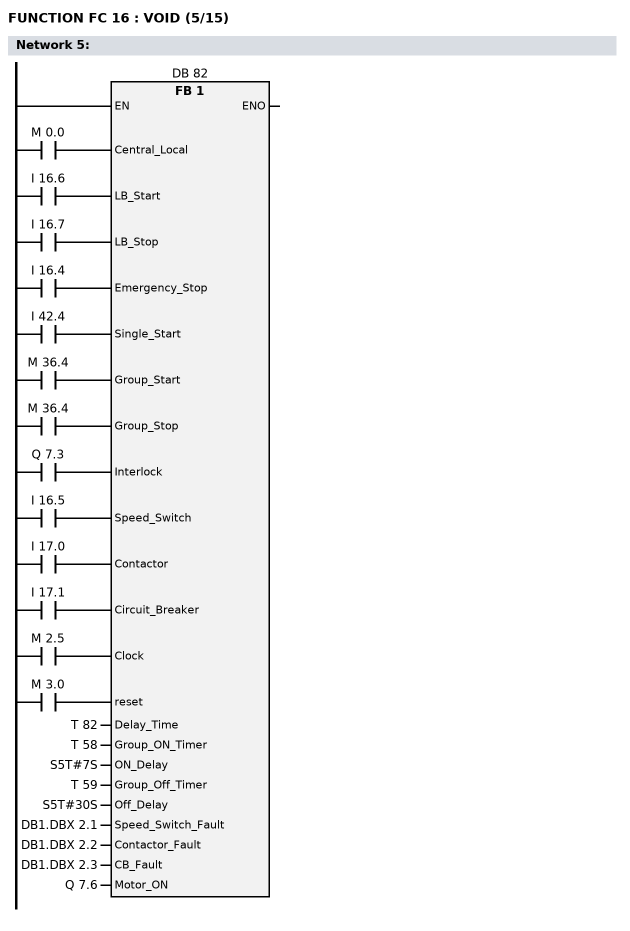

      A     M      0.0;
      =     L      0.0;
      BLD   103;
      A     I     16.6;
      =     L      0.1;
      BLD   103;
      A     I     16.7;
      =     L      0.2;
      BLD   103;
      A     I     16.4;
      =     L      0.3;
      BLD   103;
      A     I     42.4;
      =     L      0.4;
      BLD   103;
      A     M     36.4;
      =     L      0.5;
      BLD   103;
      A     M     36.4;
      =     L      0.6;
      BLD   103;
      A     Q      7.3;
      =     L      0.7;
      BLD   103;
      A     I     16.5;
      =     L      1.0;
      BLD   103;
      A     I     17.0;
      =     L      1.1;
      BLD   103;
      A     I     17.1;
      =     L      1.2;
      BLD   103;
      A     M      2.5;
      =     L      1.3;
      BLD   103;
      A     M      3.0;
      =     L      1.4;
      BLD   103;
      CALL FB     1 , DB    82 (
           Central_Local            := L      0.0,
           LB_Start                 := L      0.1,
           LB_Stop                  := L      0.2,
           Emergency_Stop           := L      0.3,
           Single_Start             := L      0.4,
           Group_Start              := L      0.5,
           Group_Stop               := L      0.6,
           Interlock                := L      0.7,
           Speed_Switch             := L      1.0,
           Contactor                := L      1.1,
           Circuit_Breaker          := L      1.2,
           Clock                    := L      1.3,
           reset                    := L      1.4,
           Delay_Time               := T     82,
           Group_ON_Timer           := T     58,
           ON_Delay                 := S5T#7S,
           Group_Off_Timer          := T     59,
           Off_Delay                := S5T#30S,
           Speed_Switch_Fault       := DB1.DBX    2.1,
           Contactor_Fault          := DB1.DBX    2.2,
           CB_Fault                 := DB1.DBX    2.3,
           Motor_ON                 := Q      7.6);
      NOP   0;
NETWORK
TITLE =
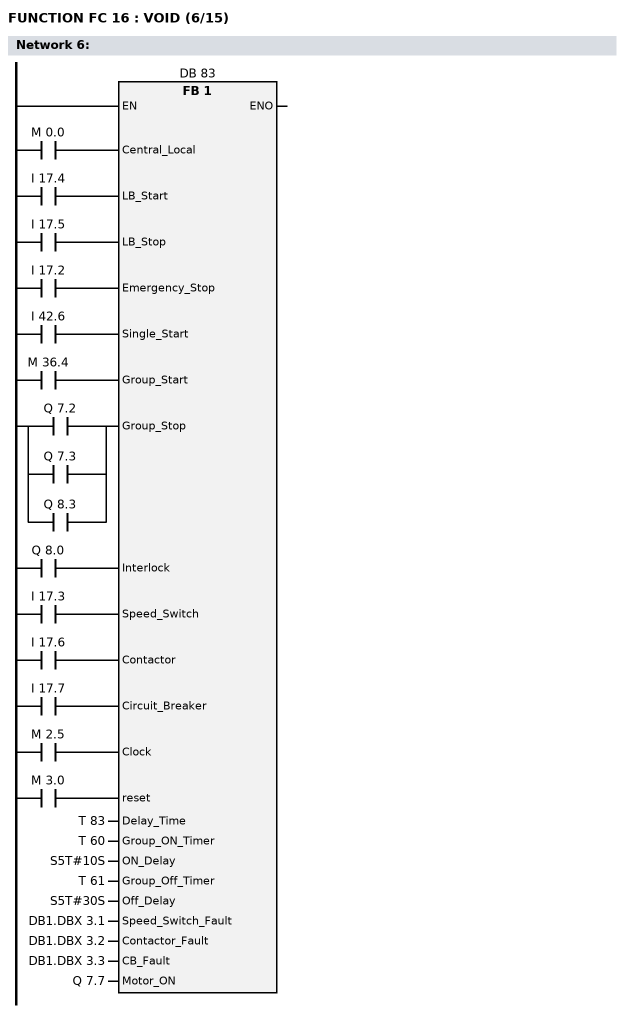

      A     M      0.0;
      =     L      0.0;
      BLD   103;
      A     I     17.4;
      =     L      0.1;
      BLD   103;
      A     I     17.5;
      =     L      0.2;
      BLD   103;
      A     I     17.2;
      =     L      0.3;
      BLD   103;
      A     I     42.6;
      =     L      0.4;
      BLD   103;
      A     M     36.4;
      =     L      0.5;
      BLD   103;
      A(    ;
      O     Q      7.2;
      O     Q      7.3;
      O     Q      8.3;
      )     ;
      =     L      0.6;
      BLD   103;
      A     Q      8.0;
      =     L      0.7;
      BLD   103;
      A     I     17.3;
      =     L      1.0;
      BLD   103;
      A     I     17.6;
      =     L      1.1;
      BLD   103;
      A     I     17.7;
      =     L      1.2;
      BLD   103;
      A     M      2.5;
      =     L      1.3;
      BLD   103;
      A     M      3.0;
      =     L      1.4;
      BLD   103;
      CALL FB     1 , DB    83 (
           Central_Local            := L      0.0,
           LB_Start                 := L      0.1,
           LB_Stop                  := L      0.2,
           Emergency_Stop           := L      0.3,
           Single_Start             := L      0.4,
           Group_Start              := L      0.5,
           Group_Stop               := L      0.6,
           Interlock                := L      0.7,
           Speed_Switch             := L      1.0,
           Contactor                := L      1.1,
           Circuit_Breaker          := L      1.2,
           Clock                    := L      1.3,
           reset                    := L      1.4,
           Delay_Time               := T     83,
           Group_ON_Timer           := T     60,
           ON_Delay                 := S5T#10S,
           Group_Off_Timer          := T     61,
           Off_Delay                := S5T#30S,
           Speed_Switch_Fault       := DB1.DBX    3.1,
           Contactor_Fault          := DB1.DBX    3.2,
           CB_Fault                 := DB1.DBX    3.3,
           Motor_ON                 := Q      7.7);
      NOP   0;
NETWORK
TITLE =
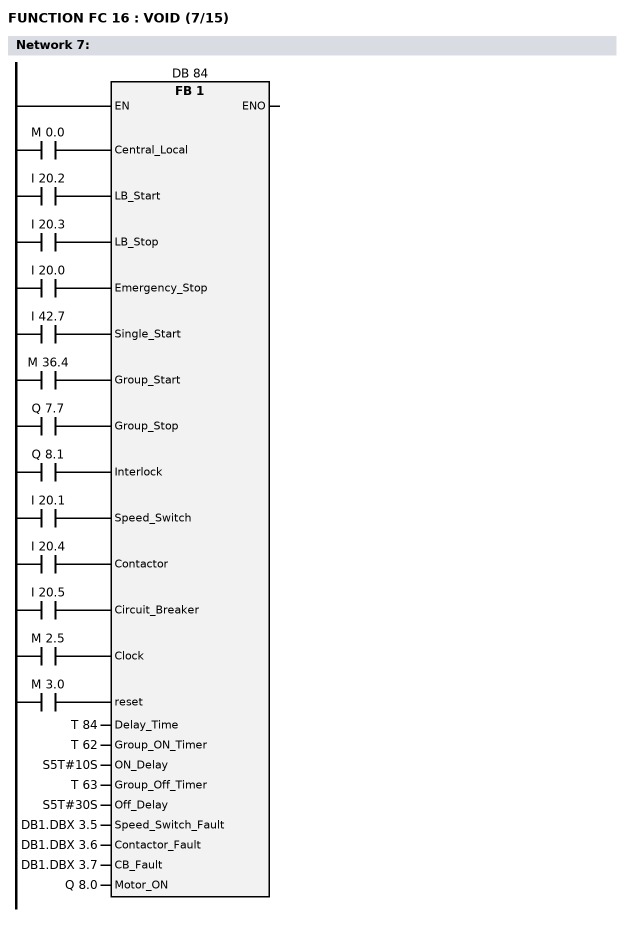

      A     M      0.0;
      =     L      0.0;
      BLD   103;
      A     I     20.2;
      =     L      0.1;
      BLD   103;
      A     I     20.3;
      =     L      0.2;
      BLD   103;
      A     I     20.0;
      =     L      0.3;
      BLD   103;
      A     I     42.7;
      =     L      0.4;
      BLD   103;
      A     M     36.4;
      =     L      0.5;
      BLD   103;
      A     Q      7.7;
      =     L      0.6;
      BLD   103;
      A     Q      8.1;
      =     L      0.7;
      BLD   103;
      A     I     20.1;
      =     L      1.0;
      BLD   103;
      A     I     20.4;
      =     L      1.1;
      BLD   103;
      A     I     20.5;
      =     L      1.2;
      BLD   103;
      A     M      2.5;
      =     L      1.3;
      BLD   103;
      A     M      3.0;
      =     L      1.4;
      BLD   103;
      CALL FB     1 , DB    84 (
           Central_Local            := L      0.0,
           LB_Start                 := L      0.1,
           LB_Stop                  := L      0.2,
           Emergency_Stop           := L      0.3,
           Single_Start             := L      0.4,
           Group_Start              := L      0.5,
           Group_Stop               := L      0.6,
           Interlock                := L      0.7,
           Speed_Switch             := L      1.0,
           Contactor                := L      1.1,
           Circuit_Breaker          := L      1.2,
           Clock                    := L      1.3,
           reset                    := L      1.4,
           Delay_Time               := T     84,
           Group_ON_Timer           := T     62,
           ON_Delay                 := S5T#10S,
           Group_Off_Timer          := T     63,
           Off_Delay                := S5T#30S,
           Speed_Switch_Fault       := DB1.DBX    3.5,
           Contactor_Fault          := DB1.DBX    3.6,
           CB_Fault                 := DB1.DBX    3.7,
           Motor_ON                 := Q      8.0);
      NOP   0;
NETWORK
TITLE =
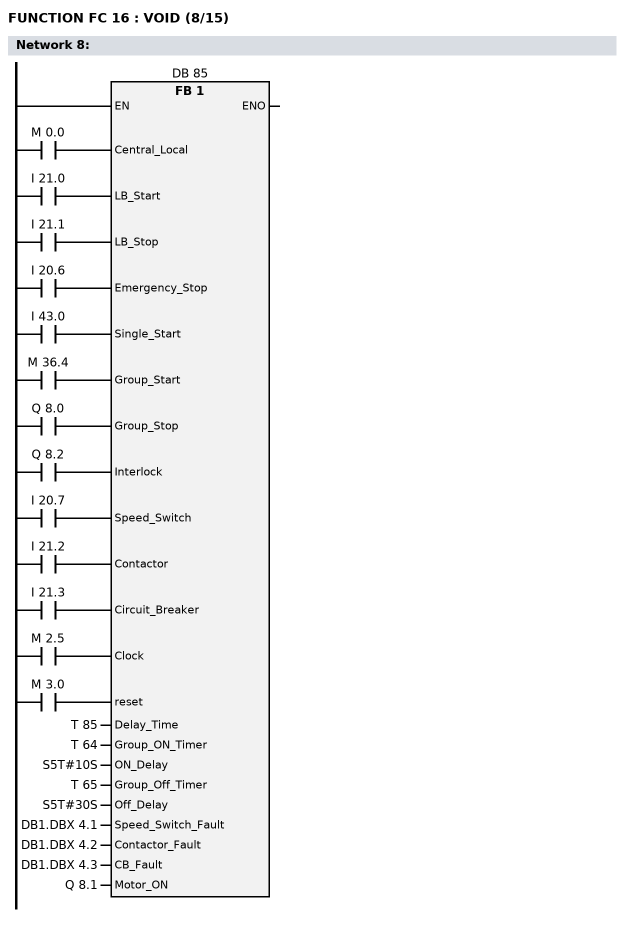

      A     M      0.0;
      =     L      0.0;
      BLD   103;
      A     I     21.0;
      =     L      0.1;
      BLD   103;
      A     I     21.1;
      =     L      0.2;
      BLD   103;
      A     I     20.6;
      =     L      0.3;
      BLD   103;
      A     I     43.0;
      =     L      0.4;
      BLD   103;
      A     M     36.4;
      =     L      0.5;
      BLD   103;
      A     Q      8.0;
      =     L      0.6;
      BLD   103;
      A     Q      8.2;
      =     L      0.7;
      BLD   103;
      A     I     20.7;
      =     L      1.0;
      BLD   103;
      A     I     21.2;
      =     L      1.1;
      BLD   103;
      A     I     21.3;
      =     L      1.2;
      BLD   103;
      A     M      2.5;
      =     L      1.3;
      BLD   103;
      A     M      3.0;
      =     L      1.4;
      BLD   103;
      CALL FB     1 , DB    85 (
           Central_Local            := L      0.0,
           LB_Start                 := L      0.1,
           LB_Stop                  := L      0.2,
           Emergency_Stop           := L      0.3,
           Single_Start             := L      0.4,
           Group_Start              := L      0.5,
           Group_Stop               := L      0.6,
           Interlock                := L      0.7,
           Speed_Switch             := L      1.0,
           Contactor                := L      1.1,
           Circuit_Breaker          := L      1.2,
           Clock                    := L      1.3,
           reset                    := L      1.4,
           Delay_Time               := T     85,
           Group_ON_Timer           := T     64,
           ON_Delay                 := S5T#10S,
           Group_Off_Timer          := T     65,
           Off_Delay                := S5T#30S,
           Speed_Switch_Fault       := DB1.DBX    4.1,
           Contactor_Fault          := DB1.DBX    4.2,
           CB_Fault                 := DB1.DBX    4.3,
           Motor_ON                 := Q      8.1);
      NOP   0;
NETWORK
TITLE =
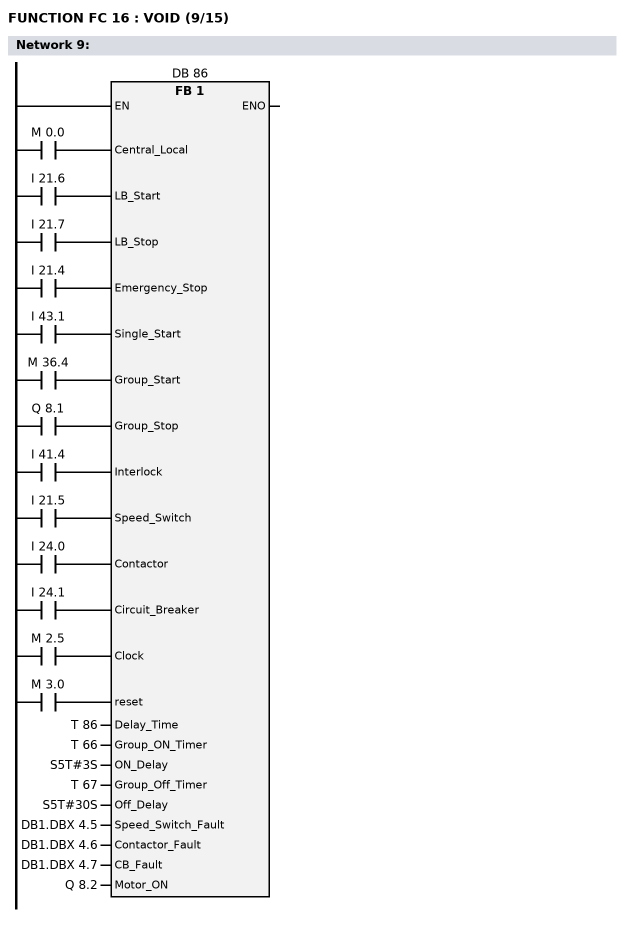

      A     M      0.0;
      =     L      0.0;
      BLD   103;
      A     I     21.6;
      =     L      0.1;
      BLD   103;
      A     I     21.7;
      =     L      0.2;
      BLD   103;
      A     I     21.4;
      =     L      0.3;
      BLD   103;
      A     I     43.1;
      =     L      0.4;
      BLD   103;
      A     M     36.4;
      =     L      0.5;
      BLD   103;
      A     Q      8.1;
      =     L      0.6;
      BLD   103;
      A     I     41.4;
      =     L      0.7;
      BLD   103;
      A     I     21.5;
      =     L      1.0;
      BLD   103;
      A     I     24.0;
      =     L      1.1;
      BLD   103;
      A     I     24.1;
      =     L      1.2;
      BLD   103;
      A     M      2.5;
      =     L      1.3;
      BLD   103;
      A     M      3.0;
      =     L      1.4;
      BLD   103;
      CALL FB     1 , DB    86 (
           Central_Local            := L      0.0,
           LB_Start                 := L      0.1,
           LB_Stop                  := L      0.2,
           Emergency_Stop           := L      0.3,
           Single_Start             := L      0.4,
           Group_Start              := L      0.5,
           Group_Stop               := L      0.6,
           Interlock                := L      0.7,
           Speed_Switch             := L      1.0,
           Contactor                := L      1.1,
           Circuit_Breaker          := L      1.2,
           Clock                    := L      1.3,
           reset                    := L      1.4,
           Delay_Time               := T     86,
           Group_ON_Timer           := T     66,
           ON_Delay                 := S5T#3S,
           Group_Off_Timer          := T     67,
           Off_Delay                := S5T#30S,
           Speed_Switch_Fault       := DB1.DBX    4.5,
           Contactor_Fault          := DB1.DBX    4.6,
           CB_Fault                 := DB1.DBX    4.7,
           Motor_ON                 := Q      8.2);
      NOP   0;
NETWORK
TITLE =
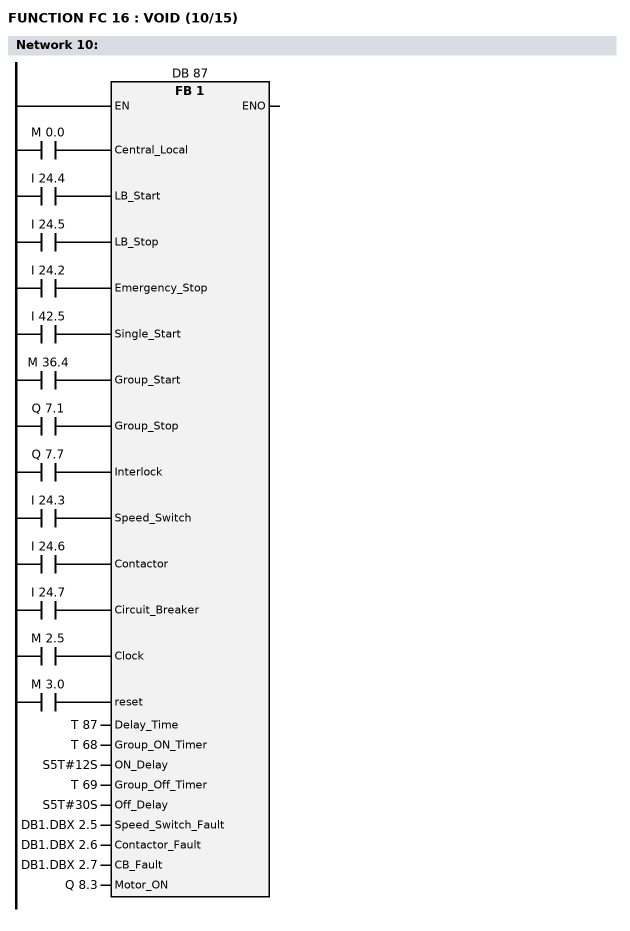

      A     M      0.0;
      =     L      0.0;
      BLD   103;
      A     I     24.4;
      =     L      0.1;
      BLD   103;
      A     I     24.5;
      =     L      0.2;
      BLD   103;
      A     I     24.2;
      =     L      0.3;
      BLD   103;
      A     I     42.5;
      =     L      0.4;
      BLD   103;
      A     M     36.4;
      =     L      0.5;
      BLD   103;
      A     Q      7.1;
      =     L      0.6;
      BLD   103;
      A     Q      7.7;
      =     L      0.7;
      BLD   103;
      A     I     24.3;
      =     L      1.0;
      BLD   103;
      A     I     24.6;
      =     L      1.1;
      BLD   103;
      A     I     24.7;
      =     L      1.2;
      BLD   103;
      A     M      2.5;
      =     L      1.3;
      BLD   103;
      A     M      3.0;
      =     L      1.4;
      BLD   103;
      CALL FB     1 , DB    87 (
           Central_Local            := L      0.0,
           LB_Start                 := L      0.1,
           LB_Stop                  := L      0.2,
           Emergency_Stop           := L      0.3,
           Single_Start             := L      0.4,
           Group_Start              := L      0.5,
           Group_Stop               := L      0.6,
           Interlock                := L      0.7,
           Speed_Switch             := L      1.0,
           Contactor                := L      1.1,
           Circuit_Breaker          := L      1.2,
           Clock                    := L      1.3,
           reset                    := L      1.4,
           Delay_Time               := T     87,
           Group_ON_Timer           := T     68,
           ON_Delay                 := S5T#12S,
           Group_Off_Timer          := T     69,
           Off_Delay                := S5T#30S,
           Speed_Switch_Fault       := DB1.DBX    2.5,
           Contactor_Fault          := DB1.DBX    2.6,
           CB_Fault                 := DB1.DBX    2.7,
           Motor_ON                 := Q      8.3);
      NOP   0;
NETWORK
TITLE =
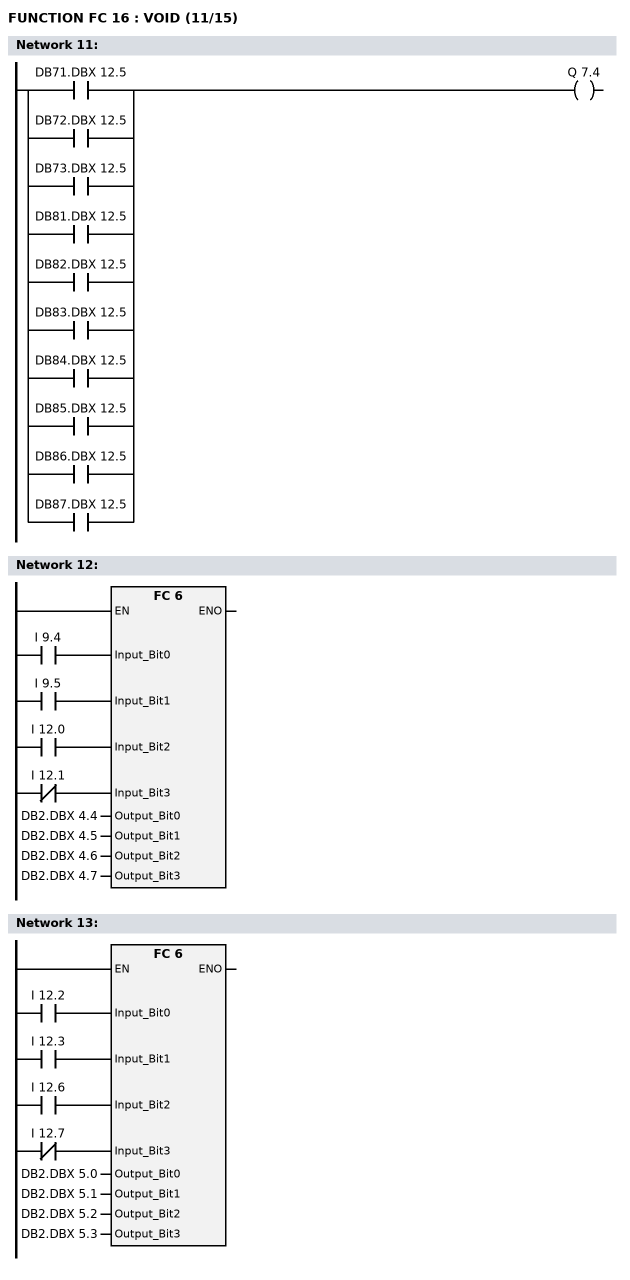

      O     DB71.DBX   12.5;
      O     DB72.DBX   12.5;
      O     DB73.DBX   12.5;
      O     DB81.DBX   12.5;
      O     DB82.DBX   12.5;
      O     DB83.DBX   12.5;
      O     DB84.DBX   12.5;
      O     DB85.DBX   12.5;
      O     DB86.DBX   12.5;
      O     DB87.DBX   12.5;
      =     Q      7.4;
NETWORK
TITLE =

      A     I      9.4;
      =     L      0.0;
      BLD   103;
      A     I      9.5;
      =     L      0.1;
      BLD   103;
      A     I     12.0;
      =     L      0.2;
      BLD   103;
      AN    I     12.1;
      =     L      0.3;
      BLD   103;
      CALL FC     6 (
           Input_Bit0               := L      0.0,
           Input_Bit1               := L      0.1,
           Input_Bit2               := L      0.2,
           Input_Bit3               := L      0.3,
           Output_Bit0              := DB2.DBX    4.4,
           Output_Bit1              := DB2.DBX    4.5,
           Output_Bit2              := DB2.DBX    4.6,
           Output_Bit3              := DB2.DBX    4.7);
      NOP   0;
NETWORK
TITLE =

      A     I     12.2;
      =     L      0.0;
      BLD   103;
      A     I     12.3;
      =     L      0.1;
      BLD   103;
      A     I     12.6;
      =     L      0.2;
      BLD   103;
      AN    I     12.7;
      =     L      0.3;
      BLD   103;
      CALL FC     6 (
           Input_Bit0               := L      0.0,
           Input_Bit1               := L      0.1,
           Input_Bit2               := L      0.2,
           Input_Bit3               := L      0.3,
           Output_Bit0              := DB2.DBX    5.0,
           Output_Bit1              := DB2.DBX    5.1,
           Output_Bit2              := DB2.DBX    5.2,
           Output_Bit3              := DB2.DBX    5.3);
      NOP   0;
NETWORK
TITLE =
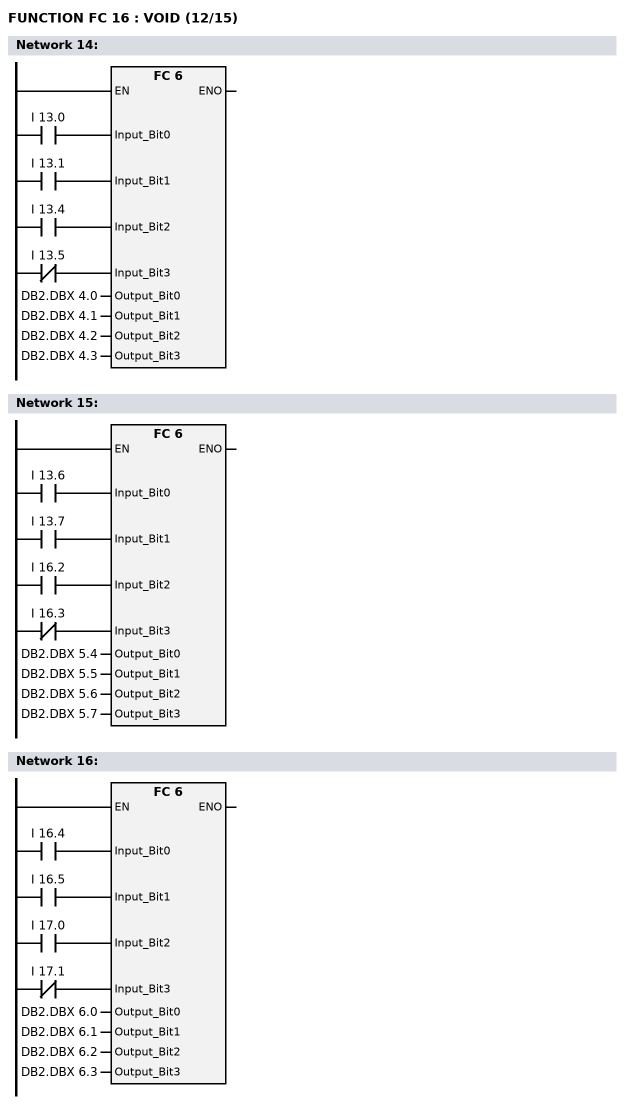

      A     I     13.0;
      =     L      0.0;
      BLD   103;
      A     I     13.1;
      =     L      0.1;
      BLD   103;
      A     I     13.4;
      =     L      0.2;
      BLD   103;
      AN    I     13.5;
      =     L      0.3;
      BLD   103;
      CALL FC     6 (
           Input_Bit0               := L      0.0,
           Input_Bit1               := L      0.1,
           Input_Bit2               := L      0.2,
           Input_Bit3               := L      0.3,
           Output_Bit0              := DB2.DBX    4.0,
           Output_Bit1              := DB2.DBX    4.1,
           Output_Bit2              := DB2.DBX    4.2,
           Output_Bit3              := DB2.DBX    4.3);
      NOP   0;
NETWORK
TITLE =

      A     I     13.6;
      =     L      0.0;
      BLD   103;
      A     I     13.7;
      =     L      0.1;
      BLD   103;
      A     I     16.2;
      =     L      0.2;
      BLD   103;
      AN    I     16.3;
      =     L      0.3;
      BLD   103;
      CALL FC     6 (
           Input_Bit0               := L      0.0,
           Input_Bit1               := L      0.1,
           Input_Bit2               := L      0.2,
           Input_Bit3               := L      0.3,
           Output_Bit0              := DB2.DBX    5.4,
           Output_Bit1              := DB2.DBX    5.5,
           Output_Bit2              := DB2.DBX    5.6,
           Output_Bit3              := DB2.DBX    5.7);
      NOP   0;
NETWORK
TITLE =

      A     I     16.4;
      =     L      0.0;
      BLD   103;
      A     I     16.5;
      =     L      0.1;
      BLD   103;
      A     I     17.0;
      =     L      0.2;
      BLD   103;
      AN    I     17.1;
      =     L      0.3;
      BLD   103;
      CALL FC     6 (
           Input_Bit0               := L      0.0,
           Input_Bit1               := L      0.1,
           Input_Bit2               := L      0.2,
           Input_Bit3               := L      0.3,
           Output_Bit0              := DB2.DBX    6.0,
           Output_Bit1              := DB2.DBX    6.1,
           Output_Bit2              := DB2.DBX    6.2,
           Output_Bit3              := DB2.DBX    6.3);
      NOP   0;
NETWORK
TITLE =
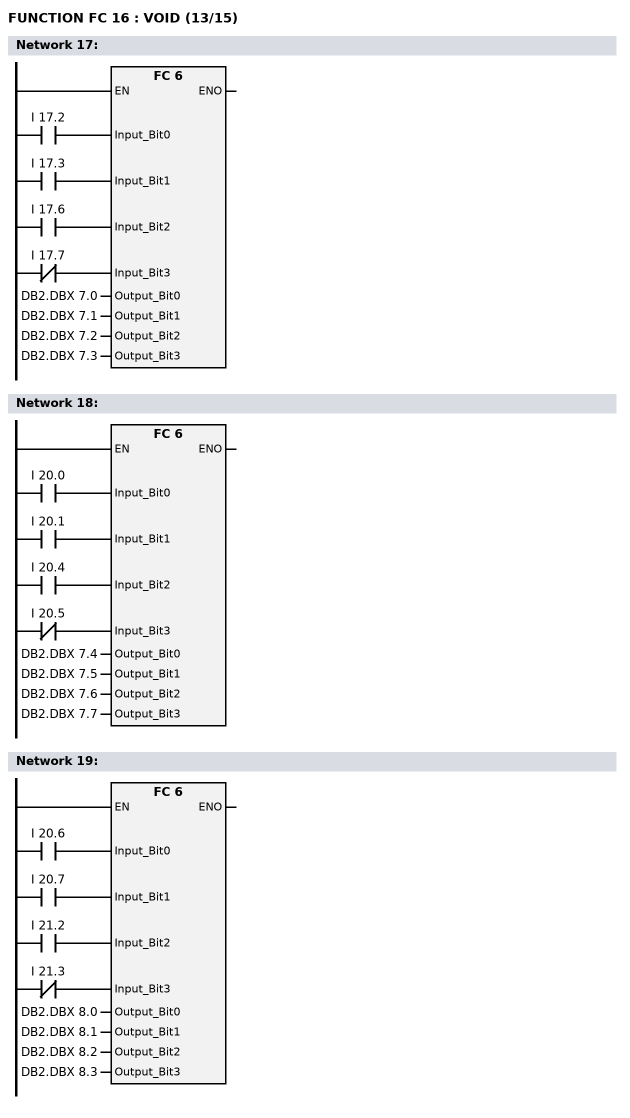

      A     I     17.2;
      =     L      0.0;
      BLD   103;
      A     I     17.3;
      =     L      0.1;
      BLD   103;
      A     I     17.6;
      =     L      0.2;
      BLD   103;
      AN    I     17.7;
      =     L      0.3;
      BLD   103;
      CALL FC     6 (
           Input_Bit0               := L      0.0,
           Input_Bit1               := L      0.1,
           Input_Bit2               := L      0.2,
           Input_Bit3               := L      0.3,
           Output_Bit0              := DB2.DBX    7.0,
           Output_Bit1              := DB2.DBX    7.1,
           Output_Bit2              := DB2.DBX    7.2,
           Output_Bit3              := DB2.DBX    7.3);
      NOP   0;
NETWORK
TITLE =

      A     I     20.0;
      =     L      0.0;
      BLD   103;
      A     I     20.1;
      =     L      0.1;
      BLD   103;
      A     I     20.4;
      =     L      0.2;
      BLD   103;
      AN    I     20.5;
      =     L      0.3;
      BLD   103;
      CALL FC     6 (
           Input_Bit0               := L      0.0,
           Input_Bit1               := L      0.1,
           Input_Bit2               := L      0.2,
           Input_Bit3               := L      0.3,
           Output_Bit0              := DB2.DBX    7.4,
           Output_Bit1              := DB2.DBX    7.5,
           Output_Bit2              := DB2.DBX    7.6,
           Output_Bit3              := DB2.DBX    7.7);
      NOP   0;
NETWORK
TITLE =

      A     I     20.6;
      =     L      0.0;
      BLD   103;
      A     I     20.7;
      =     L      0.1;
      BLD   103;
      A     I     21.2;
      =     L      0.2;
      BLD   103;
      AN    I     21.3;
      =     L      0.3;
      BLD   103;
      CALL FC     6 (
           Input_Bit0               := L      0.0,
           Input_Bit1               := L      0.1,
           Input_Bit2               := L      0.2,
           Input_Bit3               := L      0.3,
           Output_Bit0              := DB2.DBX    8.0,
           Output_Bit1              := DB2.DBX    8.1,
           Output_Bit2              := DB2.DBX    8.2,
           Output_Bit3              := DB2.DBX    8.3);
      NOP   0;
NETWORK
TITLE =
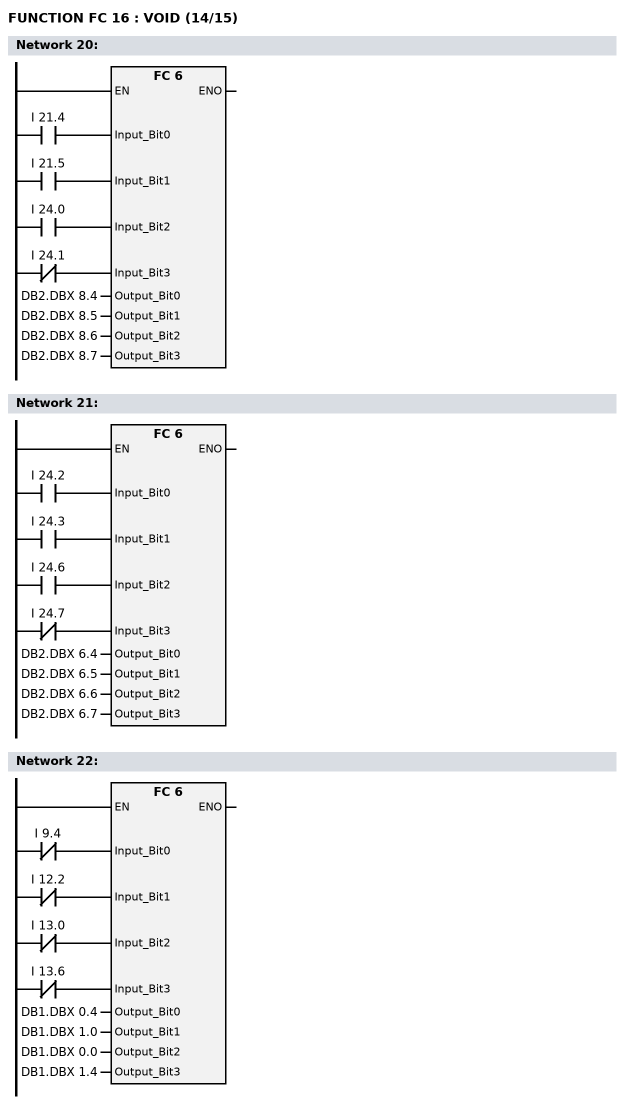

      A     I     21.4;
      =     L      0.0;
      BLD   103;
      A     I     21.5;
      =     L      0.1;
      BLD   103;
      A     I     24.0;
      =     L      0.2;
      BLD   103;
      AN    I     24.1;
      =     L      0.3;
      BLD   103;
      CALL FC     6 (
           Input_Bit0               := L      0.0,
           Input_Bit1               := L      0.1,
           Input_Bit2               := L      0.2,
           Input_Bit3               := L      0.3,
           Output_Bit0              := DB2.DBX    8.4,
           Output_Bit1              := DB2.DBX    8.5,
           Output_Bit2              := DB2.DBX    8.6,
           Output_Bit3              := DB2.DBX    8.7);
      NOP   0;
NETWORK
TITLE =

      A     I     24.2;
      =     L      0.0;
      BLD   103;
      A     I     24.3;
      =     L      0.1;
      BLD   103;
      A     I     24.6;
      =     L      0.2;
      BLD   103;
      AN    I     24.7;
      =     L      0.3;
      BLD   103;
      CALL FC     6 (
           Input_Bit0               := L      0.0,
           Input_Bit1               := L      0.1,
           Input_Bit2               := L      0.2,
           Input_Bit3               := L      0.3,
           Output_Bit0              := DB2.DBX    6.4,
           Output_Bit1              := DB2.DBX    6.5,
           Output_Bit2              := DB2.DBX    6.6,
           Output_Bit3              := DB2.DBX    6.7);
      NOP   0;
NETWORK
TITLE =

      AN    I      9.4;
      =     L      0.0;
      BLD   103;
      AN    I     12.2;
      =     L      0.1;
      BLD   103;
      AN    I     13.0;
      =     L      0.2;
      BLD   103;
      AN    I     13.6;
      =     L      0.3;
      BLD   103;
      CALL FC     6 (
           Input_Bit0               := L      0.0,
           Input_Bit1               := L      0.1,
           Input_Bit2               := L      0.2,
           Input_Bit3               := L      0.3,
           Output_Bit0              := DB1.DBX    0.4,
           Output_Bit1              := DB1.DBX    1.0,
           Output_Bit2              := DB1.DBX    0.0,
           Output_Bit3              := DB1.DBX    1.4);
      NOP   0;
NETWORK
TITLE =
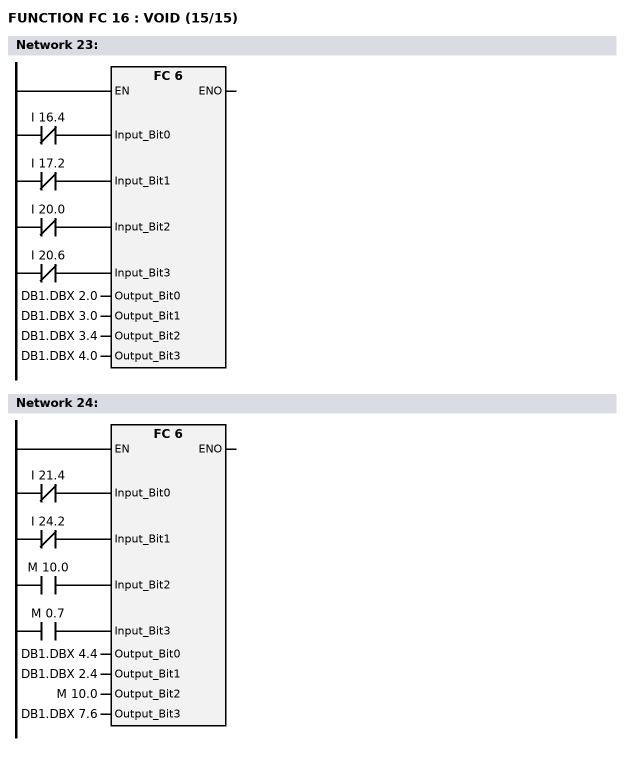

      AN    I     16.4;
      =     L      0.0;
      BLD   103;
      AN    I     17.2;
      =     L      0.1;
      BLD   103;
      AN    I     20.0;
      =     L      0.2;
      BLD   103;
      AN    I     20.6;
      =     L      0.3;
      BLD   103;
      CALL FC     6 (
           Input_Bit0               := L      0.0,
           Input_Bit1               := L      0.1,
           Input_Bit2               := L      0.2,
           Input_Bit3               := L      0.3,
           Output_Bit0              := DB1.DBX    2.0,
           Output_Bit1              := DB1.DBX    3.0,
           Output_Bit2              := DB1.DBX    3.4,
           Output_Bit3              := DB1.DBX    4.0);
      NOP   0;
NETWORK
TITLE =

      AN    I     21.4;
      =     L      0.0;
      BLD   103;
      AN    I     24.2;
      =     L      0.1;
      BLD   103;
      A     M     10.0;
      =     L      0.2;
      BLD   103;
      A     M      0.7;
      =     L      0.3;
      BLD   103;
      CALL FC     6 (
           Input_Bit0               := L      0.0,
           Input_Bit1               := L      0.1,
           Input_Bit2               := L      0.2,
           Input_Bit3               := L      0.3,
           Output_Bit0              := DB1.DBX    4.4,
           Output_Bit1              := DB1.DBX    2.4,
           Output_Bit2              := M     10.0,
           Output_Bit3              := DB1.DBX    7.6);
      NOP   0;
END_FUNCTION

FUNCTION FC 18 : VOID
TITLE =New Pulse Controller 91_8_22
VERSION : 0.1

BEGIN
NETWORK
TITLE =
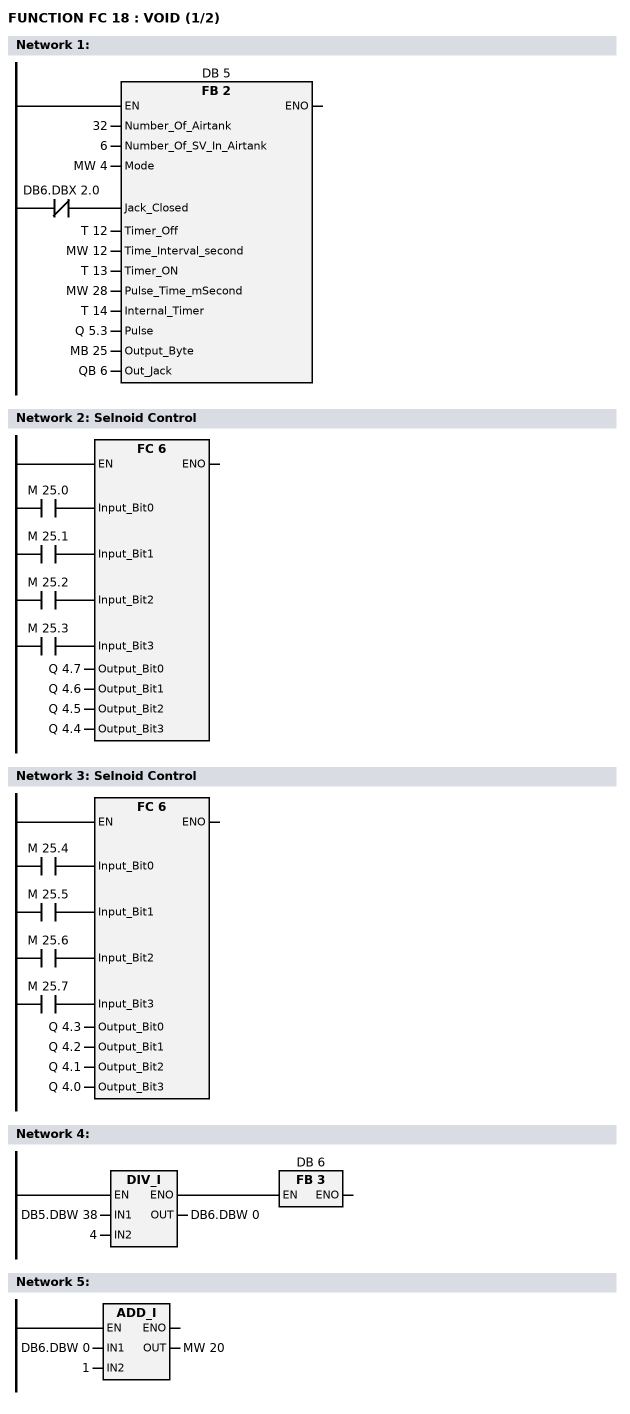

      AN    DB6.DBX    2.0;
      =     L      0.0;
      BLD   103;
      CALL FB     2 , DB     5 (
           Number_Of_Airtank        := 32,
           Number_Of_SV_In_Airtank  := 6,
           Mode                     := MW     4,
           Jack_Closed              := L      0.0,
           Timer_Off                := T     12,
           Time_Interval_second     := MW    12,
           Timer_ON                 := T     13,
           Pulse_Time_mSecond       := MW    28,
           Internal_Timer           := T     14,
           Pulse                    := Q      5.3,
           Output_Byte              := MB    25,
           Out_Jack                 := QB     6);
      NOP   0;
NETWORK
TITLE =Selnoid Control

      A     M     25.0;
      =     L      0.0;
      BLD   103;
      A     M     25.1;
      =     L      0.1;
      BLD   103;
      A     M     25.2;
      =     L      0.2;
      BLD   103;
      A     M     25.3;
      =     L      0.3;
      BLD   103;
      CALL FC     6 (
           Input_Bit0               := L      0.0,
           Input_Bit1               := L      0.1,
           Input_Bit2               := L      0.2,
           Input_Bit3               := L      0.3,
           Output_Bit0              := Q      4.7,
           Output_Bit1              := Q      4.6,
           Output_Bit2              := Q      4.5,
           Output_Bit3              := Q      4.4);
      NOP   0;
NETWORK
TITLE =Selnoid Control

      A     M     25.4;
      =     L      0.0;
      BLD   103;
      A     M     25.5;
      =     L      0.1;
      BLD   103;
      A     M     25.6;
      =     L      0.2;
      BLD   103;
      A     M     25.7;
      =     L      0.3;
      BLD   103;
      CALL FC     6 (
           Input_Bit0               := L      0.0,
           Input_Bit1               := L      0.1,
           Input_Bit2               := L      0.2,
           Input_Bit3               := L      0.3,
           Output_Bit0              := Q      4.3,
           Output_Bit1              := Q      4.2,
           Output_Bit2              := Q      4.1,
           Output_Bit3              := Q      4.0);
      NOP   0;
NETWORK
TITLE =

      A(    ;
      L     DB5.DBW   38;
      L     4;
      /I    ;
      T     DB6.DBW    0;
      AN    OV;
      SAVE  ;
      CLR   ;
      A     BR;
      )     ;
      JNB   _001;
      CALL FB     3 , DB     6 ;
_001: NOP   0;
NETWORK
TITLE =

      L     DB6.DBW    0;
      L     1;
      +I    ;
      T     MW    20;
      NOP   0;
NETWORK
TITLE =
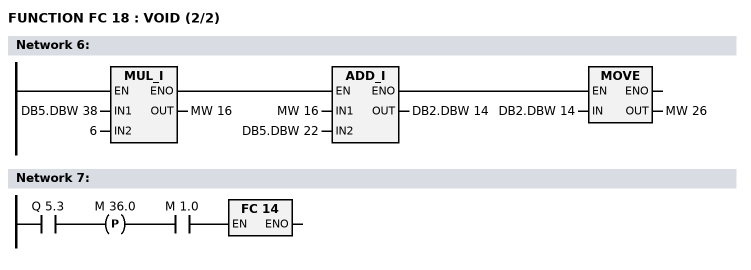

      A(    ;
      A(    ;
      L     DB5.DBW   38;
      L     6;
      *I    ;
      T     MW    16;
      AN    OV;
      SAVE  ;
      CLR   ;
      A     BR;
      )     ;
      JNB   _002;
      L     MW    16;
      L     DB5.DBW   22;
      +I    ;
      T     DB2.DBW   14;
      AN    OV;
      SAVE  ;
      CLR   ;
_002: A     BR;
      )     ;
      JNB   _003;
      L     DB2.DBW   14;
      T     MW    26;
_003: NOP   0;
NETWORK
TITLE =

      A     Q      5.3;
      FP    M     36.0;
      A     M      1.0;
      JNB   _004;
      CALL FC    14 ;
_004: NOP   0;
END_FUNCTION

ORGANIZATION_BLOCK OB 1
TITLE = "Main Program Sweep (Cycle)"
//New Version 91_8_20
VERSION : 0.1


VAR_TEMP
  OB1_EV_CLASS : BYTE ;	//Bits 0-3 = 1 (Coming event), Bits 4-7 = 1 (Event class 1)
  OB1_SCAN_1 : BYTE ;	//1 (Cold restart scan 1 of OB 1), 3 (Scan 2-n of OB 1)
  OB1_PRIORITY : BYTE ;	//Priority of OB Execution
  OB1_OB_NUMBR : BYTE ;	//1 (Organization block 1, OB1)
  OB1_RESERVED_1 : BYTE ;	//Reserved for system
  OB1_RESERVED_2 : BYTE ;	//Reserved for system
  OB1_PREV_CYCLE : INT ;	//Cycle time of previous OB1 scan (milliseconds)
  OB1_MIN_CYCLE : INT ;	//Minimum cycle time of OB1 (milliseconds)
  OB1_MAX_CYCLE : INT ;	//Maximum cycle time of OB1 (milliseconds)
  OB1_DATE_TIME : DATE_AND_TIME ;	//Date and time OB1 started
END_VAR
BEGIN
NETWORK
TITLE =
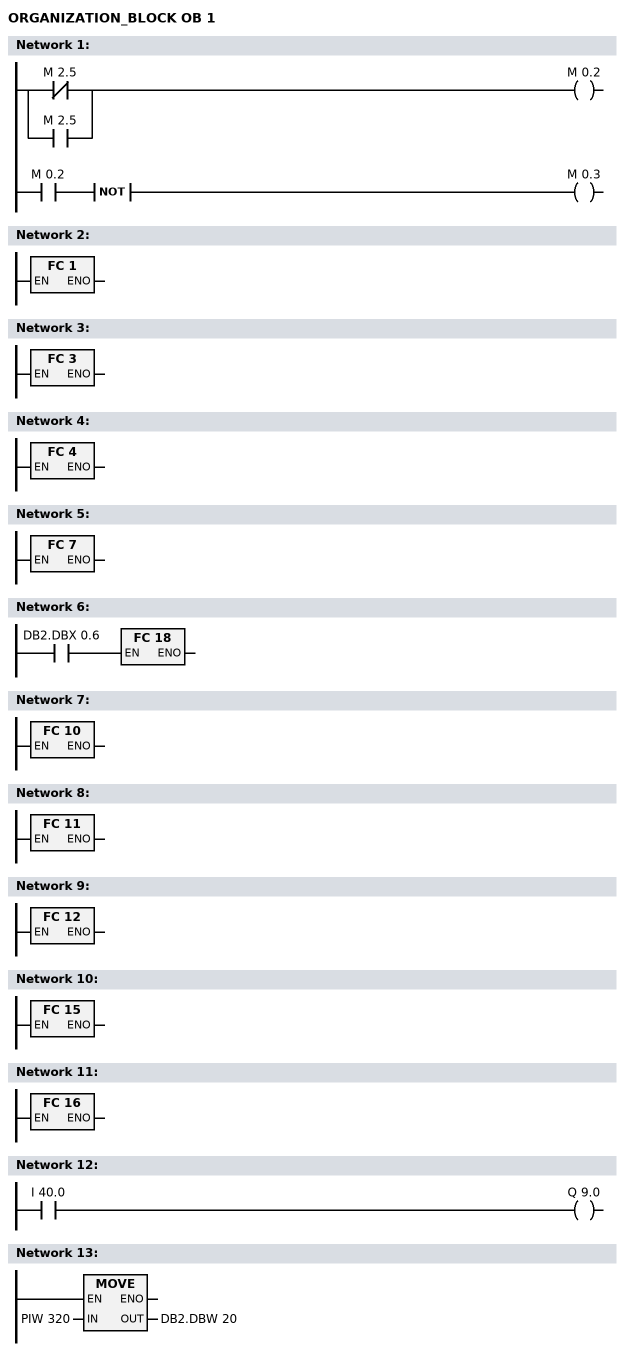

      A(    ;
      ON    M      2.5;
      O     M      2.5;
      )     ;
      =     M      0.2;
      A     M      0.2;
      NOT   ;
      =     M      0.3;
NETWORK
TITLE =

      CALL FC     1 ;
      NOP   0;
NETWORK
TITLE =

      CALL FC     3 ;
      NOP   0;
NETWORK
TITLE =

      CALL FC     4 ;
      NOP   0;
NETWORK
TITLE =

      CALL FC     7 ;
      NOP   0;
NETWORK
TITLE =

      A     DB2.DBX    0.6;
      JNB   _001;
      CALL FC    18 ;
_001: NOP   0;
NETWORK
TITLE =

      CALL FC    10 ;
      NOP   0;
NETWORK
TITLE =

      CALL FC    11 ;
      NOP   0;
NETWORK
TITLE =

      CALL FC    12 ;
      NOP   0;
NETWORK
TITLE =

      CALL FC    15 ;
      NOP   0;
NETWORK
TITLE =

      CALL FC    16 ;
      NOP   0;
NETWORK
TITLE =

      A     I     40.0;
      =     Q      9.0;
NETWORK
TITLE =

      L     PIW  320;
      T     DB2.DBW   20;
      NOP   0;
END_ORGANIZATION_BLOCK

ORGANIZATION_BLOCK OB 82
VERSION : 0.1


VAR_TEMP
  TEMP0 : BYTE ;
  TEMP1 : BYTE ;
  TEMP2 : BYTE ;
  TEMP3 : BYTE ;
  TEMP4 : BYTE ;
  TEMP5 : BYTE ;
  TEMP6 : WORD ;
  TEMP7 : BOOL ;
  TEMP8 : BOOL ;
  TEMP9 : BOOL ;
  TEMP10 : BOOL ;
  TEMP11 : BOOL ;
  TEMP12 : BOOL ;
  TEMP13 : BOOL ;
  TEMP14 : BOOL ;
  TEMP15 : BYTE ;
  TEMP16 : BOOL ;
  TEMP17 : BOOL ;
  TEMP18 : BOOL ;
  TEMP19 : BOOL ;
  TEMP20 : BOOL ;
  TEMP21 : BOOL ;
  TEMP22 : BOOL ;
  TEMP23 : BOOL ;
  TEMP24 : BOOL ;
  TEMP25 : BOOL ;
  TEMP26 : BOOL ;
  TEMP27 : BOOL ;
  TEMP28 : BOOL ;
  TEMP29 : BOOL ;
  TEMP30 : BOOL ;
  TEMP31 : BOOL ;
  TEMP32 : DATE_AND_TIME ;
END_VAR
BEGIN
END_ORGANIZATION_BLOCK

ORGANIZATION_BLOCK OB 85
TITLE = "Organization Block (OB) Not Loaded Fault"
VERSION : 0.1


VAR_TEMP
  OB85_EV_CLASS : BYTE ;	//16#35 Event class 3
  OB85_FLT_ID : BYTE ;	//16#XX, Fault identification code
  OB85_PRIORITY : BYTE ;	//Priority of OB Execution
  OB85_OB_NUMBR : BYTE ;	//85 (Organization block 85, OB85)
  OB85_RESERVED_1 : BYTE ;	//Reserved for system
  OB85_RESERVED_2 : BYTE ;	//Reserved for system
  OB85_RESERVED_3 : INT ;	//Reserved for system
  OB85_ERR_EV_CLASS : BYTE ;	//Class of event causing error
  OB85_ERR_EV_NUM : BYTE ;	//Number of event causing error
  OB85_OB_PRIOR : BYTE ;	//Priority of OB causing error
  OB85_OB_NUM : BYTE ;	//Number of OB causing error
  OB85_DATE_TIME : DATE_AND_TIME ;	//Date and time OB85 started
END_VAR
BEGIN
END_ORGANIZATION_BLOCK

ORGANIZATION_BLOCK OB 86
VERSION : 0.1


VAR_TEMP
  TEMP0 : BYTE ;
  TEMP1 : BYTE ;
  TEMP2 : BYTE ;
  TEMP3 : BYTE ;
  TEMP4 : BYTE ;
  TEMP5 : BYTE ;
  TEMP6 : WORD ;
 // TEMP7 : ARRAY  [0 .. 31 ] OF BOOL ;
  TEMP8 : DATE_AND_TIME ;
END_VAR
BEGIN
END_ORGANIZATION_BLOCK

ORGANIZATION_BLOCK OB 87
TITLE = "Communication Fault"
VERSION : 0.1


VAR_TEMP
  OB87_EV_CLASS : BYTE ;	//16#39 Event class 3
  OB87_FLT_ID : BYTE ;	//16#XX, Fault identifcation code
  OB87_PRIORITY : BYTE ;	//Priority of OB Execution
  OB87_OB_NUMBR : BYTE ;	//87 (Organization block 87, OB87)
  OB87_RESERVED_1 : BYTE ;	//Reserved for system
  OB87_RESERVED_2 : BYTE ;	//Reserved for system
  OB87_RESERVED_3 : WORD ;	//Reserved for system
  OB87_RESERVED_4 : DWORD ;	//Reserved for system
  OB87_DATE_TIME : DATE_AND_TIME ;	//Date and time OB87 started
END_VAR
BEGIN
END_ORGANIZATION_BLOCK

ORGANIZATION_BLOCK OB 121
TITLE = "Programming Error"
VERSION : 0.1


VAR_TEMP
  OB121_EV_CLASS : BYTE ;	//16#25, Event class 2, Entering event state, Internal fault event
  OB121_SW_FLT : BYTE ;	//16#XX Software programming fault
  OB121_PRIORITY : BYTE ;	//Priority of OB Execution
  OB121_OB_NUMBR : BYTE ;	//121 (Organization block 121, OB121)
  OB121_BLK_TYPE : BYTE ;	//16#88/8A/8B/8C/8E Type of block fault occured in
  OB121_RESERVED_1 : BYTE ;	//Reserved for system
  OB121_FLT_REG : WORD ;	//16#XX Specific register that caused fault
  OB121_BLK_NUM : WORD ;	//Number of block that programming fault occured in
  OB121_PRG_ADDR : WORD ;	//Address in block where programming fault occured
  OB121_DATE_TIME : DATE_AND_TIME ;	//Date and time OB121 started
END_VAR
BEGIN
END_ORGANIZATION_BLOCK

ORGANIZATION_BLOCK OB 122
VERSION : 0.1


VAR_TEMP
  TEMP0 : BYTE ;
  TEMP1 : BYTE ;
  TEMP2 : BYTE ;
  TEMP3 : BYTE ;
  TEMP4 : BYTE ;
  TEMP5 : BYTE ;
  TEMP6 : WORD ;
  TEMP7 : WORD ;
  TEMP8 : WORD ;
  TEMP9 : DATE_AND_TIME ;
END_VAR
BEGIN
END_ORGANIZATION_BLOCK

